(* PLC project GalvPLC, Beckhoff Automation GmbH TwinCAT PLC Control 3.5.19.61 *)
(* stored: creationDateTime 2026-02-19T00:33:13.1078117, modificationDateTime 2026-02-19T00:33:13.1312004 *)

{attribute 'qualified_only'}
{attribute 'strict'}
{attribute 'to_string'}
TYPE EN_DISP_MSGTYPE :
(
	none := 0,
	precheck,
	finishedOk,
	finishedWarn,
	StopReq
);
END_TYPE

{attribute 'qualified_only'}
{attribute 'strict'}
{attribute 'to_string'}
TYPE EN_DISP_POOL_STATE :
(
	empty := 0,
	newForm,
	formLoaded,
	pause,
	error,
	warning,
	precoating,
	coating,
	enchase,
	mount,
	finished
);
END_TYPE

TYPE ST_DISP_DATA :
STRUCT
	dtCurrentTime: DATE_AND_TIME;
	bGlobalErr: BOOL;
	bAckErr: BOOL;
	aPools: ARRAY [1..1] OF ST_DISP_POOL;
END_STRUCT
END_TYPE

TYPE ST_DISP_ERRORS :
STRUCT
	stGlobalErrors: ST_DISP_GOLBAL_ERRORS;
	aPoolErrors: ARRAY[1..1] OF ST_DISP_POOL_ERRORS;	
END_STRUCT
END_TYPE

TYPE ST_DISP_GOLBAL_ERRORS :
STRUCT
	bEmergStop: BOOL;
	bDriveSupplyErr: BOOL;
	bTempWarn: BOOL;
	bTempErr: BOOL;
END_STRUCT
END_TYPE

TYPE ST_DISP_MIXER :
STRUCT
	fPower: REAL;
	bManu: BOOL;
END_STRUCT
END_TYPE

TYPE ST_DISP_MIXER_ERRORS :
STRUCT
	bDriveWarn: BOOL;
	bDriveErr: BOOL;
	bOverloadErr: BOOL;
	bUnderloadWarn: BOOL;
	bVeloErr: BOOL;
END_STRUCT
END_TYPE

TYPE ST_DISP_MSG :
STRUCT
	eType: EN_DISP_MSGTYPE;	
	bEnableOk: BOOL;
	bEnableCancel: BOOL;
	bOk: BOOL;
	bCancel: BOOL;
END_STRUCT
END_TYPE

TYPE ST_DISP_POOL :
STRUCT
	sPoolName: STRING(31);
	nFormulaId: DWORD;
	sFormulaName: STRING(31);
	eState: EN_DISP_POOL_STATE;
	fTemp: REAL;
	fCurrent: REAL;
	fVoltage: REAL;
	fTiltPos: REAL;
	fTiltVelo: REAL;
	fSectPos: REAL;
	fSectVelo: REAL;
	fLeakPress: REAL;
	tProcTimeTotal: TIME;
	tProcTimeRem: TIME;
	tPhaseTimeTotal: TIME;
	tPhaseTimeRem: TIME;
	nShiftCurr: WORD;
	nShiftCount: WORD;
	nRepeatCurr: WORD;
	nRepeatCount: WORD;

	fTempSetpoint: REAL;
	bPumpOnIdle: BOOL;
	tMixerTimeManual: TIME;
	tMixerTimeAuto: TIME; (* TODO: pool param/Form ? *)

	bManuEnable: BOOL;

	bFormStart: BOOL;
	bFormStop: BOOL;
	bFormPause: BOOL;
	bTiltJogPos: BOOL;
	bTiltJogNeg: BOOL;
	bSectJogNeg: BOOL;

	stMsg: ST_DISP_MSG;

	aMixers: ARRAY [1..4] OF ST_DISP_MIXER;
END_STRUCT
END_TYPE

TYPE ST_DISP_POOL_ERRORS :
STRUCT
	bHeaterTempWarn: BOOL;
	bHeaterSensorErr: BOOL;
	bHeaterSafetyErr: BOOL;
	bTiltDriveWarn: BOOL;
	bTiltDriveErr: BOOL;
	bTiltFollowingErr: BOOL;
	bSectDriveWarn: BOOL;
	bSectDriveErr: BOOL;
	bSectFollowingErr: BOOL;
	bPsComErr: BOOL;
	bPsTempWarn: BOOL;
	bPsTempErr: BOOL;
	bPsCurrErr: BOOL;
	bPsVoltErr: BOOL;

	aMixerErrors: ARRAY [1..4] OF ST_DISP_MIXER_ERRORS;
END_STRUCT
END_TYPE

(* global variable list DISPLAY_DATA *)
{attribute 'qualified_only'}
VAR_GLOBAL
	stData: ST_DISP_DATA;
	stErrors: ST_DISP_ERRORS;
END_VAR
